(* PLC project  *)

CONFIGURATION StepIM_Conv
END_CONFIGURATION
